TYPE ST_ClampTorqueConfig :
STRUCT
    fTargetTorquePercent : LREAL;
    fMaxAbsTorquePercent : LREAL;
    fTorqueRampPercentPerSecond : LREAL;
    fVelocityLimitHigh : LREAL;
    fVelocityLimitLow : LREAL;
    fReachedMinAbsTorquePercent : LREAL;
    tReachedStableTime : TIME;
    tTorqueBuildTimeout : TIME;
    tModeSwitchTimeout : TIME;
END_STRUCT
END_TYPE

(* stored: Version 1.1.0.1, ProductVersion 3.1.4026.20
   DUT ST_ClampTorqueConfig: Id {86001ccc-2114-434d-8bcf-d100837e4bff} *)
